{attribute 'qualified_only'}
VAR_GLOBAL CONSTANT
	MaxMotionTasks : UDINT := 10;
END_VAR

(* stored: Version 1.1.0.1, ProductVersion 3.1.4026.18
   GVL ApplicationBaseMotionParameterNc2: Id {148acb86-38c9-4166-99d7-19cdb7d01c87}, ParameterList True *)
